# EPICS substitutions: support/ebrick/2-2-3/iocBoot/iocebrick/serialLink.substitutions
file "../../db/serialLink.db"
{
pattern
{P,     R,        PORT}
{ebrick:,  Slp:,     SLP}
}

file "../../db/serialLinkBC059.db"
{
pattern
{P,     R}
{ebrick:,  Slp:}
}
